// S11: the GRAPH chain's single-instance DB (a GRAPH FB cannot be a multi-instance).
DATA_BLOCK "S11Graph"
{ S7_Optimized_Access := 'TRUE' }
VERSION : 0.1
NON_RETAIN
"FB_SpkAutoGraph"

BEGIN

END_DATA_BLOCK
